(* Logix 5000 project; controller Amvex_Thorpe_Flowmeter vendor 1 type 14 code 106 rev 33.13; software revision 33.01; part 14 of 16 *)
(* tags used below, declared in another part *)
   Barcode_Result_DATA : SINT[128];
   HMI_Counter_ONS : BOOL;
   IV3_Prog_AOI : IvSwichPrgoram;
   Part_count : DINT;
   Prog_Switch_ons : BOOL;
   SR_Read_Request : BOOL;
   Test : Connect;
   Alicat_Status_ONS : BOOL[32];
   Barcode_timeout : TIMER;
   Cycle_Count_Ctr : COUNTER;
   Cycle_Count_ONS : BOOL;
   Cycle_Time_ONS : BOOL;
   FIRST_SCAN : BOOL;
   HMI : HMI_Temp;
   MCP : MCP;
   RCP1 : RCP1;
   RCP1_00 : UDT_ID0;
   Safety_OK : BOOL;
   Temp_Cycle_Time_Current : REAL;
   Temp_Cycle_Time_Last : REAL;
   Temp_Cycle_Timer : TIMER;
(* MCP_Main, continued *)

ROUTINE R09_IV3_VISION   (* ladder *)
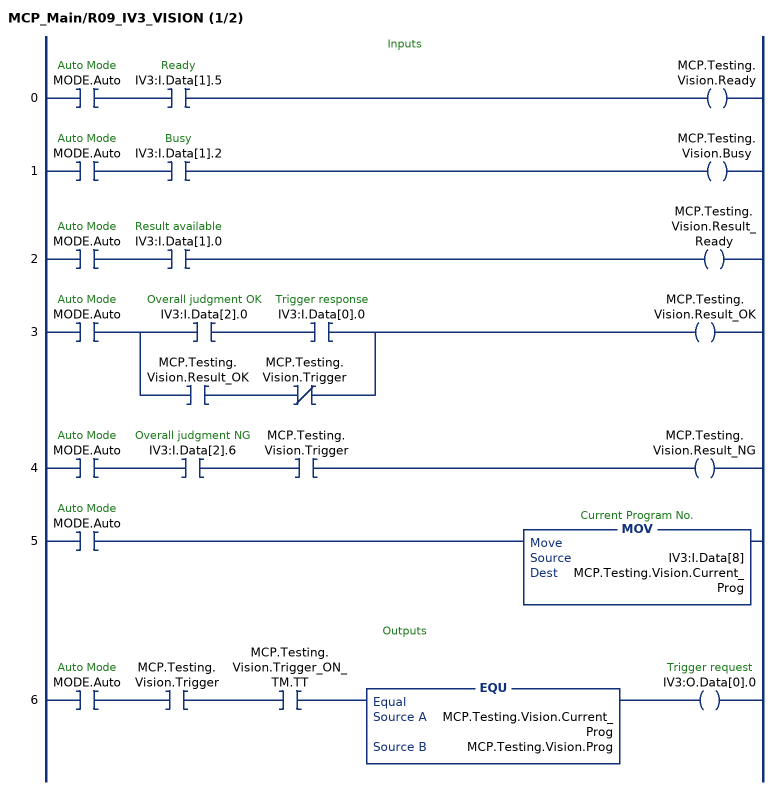
   // Inputs
   0: XIC(MODE.Auto)XIC(IV3:I.Data[1].5)OTE(MCP.Testing.Vision.Ready);
   1: XIC(MODE.Auto)XIC(IV3:I.Data[1].2)OTE(MCP.Testing.Vision.Busy);
   2: XIC(MODE.Auto)XIC(IV3:I.Data[1].0)OTE(MCP.Testing.Vision.Result_Ready);
   3: XIC(MODE.Auto)[XIC(IV3:I.Data[2].0) XIC(IV3:I.Data[0].0) ,XIC(MCP.Testing.Vision.Result_OK) XIO(MCP.Testing.Vision.Trigger) ]OTE(MCP.Testing.Vision.Result_OK);
   4: XIC(MODE.Auto)XIC(IV3:I.Data[2].6)XIC(MCP.Testing.Vision.Trigger)OTE(MCP.Testing.Vision.Result_NG);
   5: XIC(MODE.Auto)MOV(IV3:I.Data[8],MCP.Testing.Vision.Current_Prog);
   // Outputs
   6: XIC(MODE.Auto)XIC(MCP.Testing.Vision.Trigger)XIC(MCP.Testing.Vision.Trigger_ON_TM.TT)EQU(MCP.Testing.Vision.Current_Prog,MCP.Testing.Vision.Prog)OTE(IV3:O.Data[0].0);
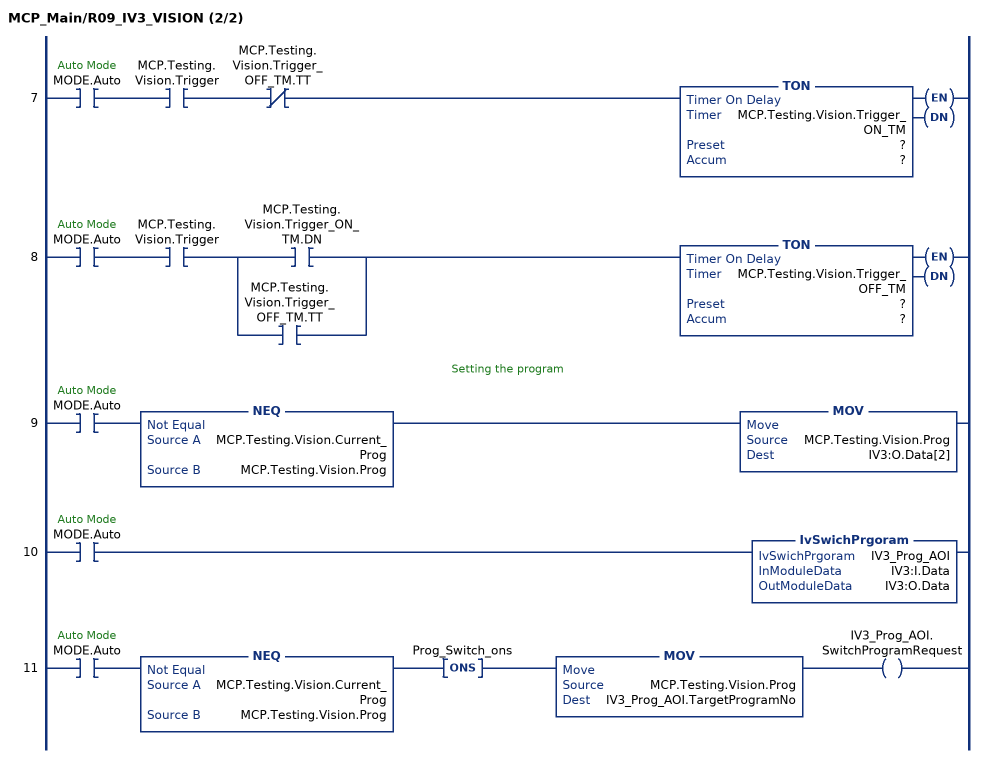
   7: XIC(MODE.Auto)XIC(MCP.Testing.Vision.Trigger)XIO(MCP.Testing.Vision.Trigger_OFF_TM.TT)TON(MCP.Testing.Vision.Trigger_ON_TM,?,?);
   8: XIC(MODE.Auto)XIC(MCP.Testing.Vision.Trigger)[XIC(MCP.Testing.Vision.Trigger_ON_TM.DN) ,XIC(MCP.Testing.Vision.Trigger_OFF_TM.TT) ]TON(MCP.Testing.Vision.Trigger_OFF_TM,?,?);
   // Setting the program
   9: XIC(MODE.Auto)NEQ(MCP.Testing.Vision.Current_Prog,MCP.Testing.Vision.Prog)MOV(MCP.Testing.Vision.Prog,IV3:O.Data[2]);
   10: XIC(MODE.Auto)IvSwichPrgoram(IV3_Prog_AOI,IV3:I.Data,IV3:O.Data);
   11: XIC(MODE.Auto)NEQ(MCP.Testing.Vision.Current_Prog,MCP.Testing.Vision.Prog)ONS(Prog_Switch_ons)MOV(MCP.Testing.Vision.Prog,IV3_Prog_AOI.TargetProgramNo)OTE(IV3_Prog_AOI.SwitchProgramRequest);
END_ROUTINE

ROUTINE R10_BARCODE   (* ladder *)
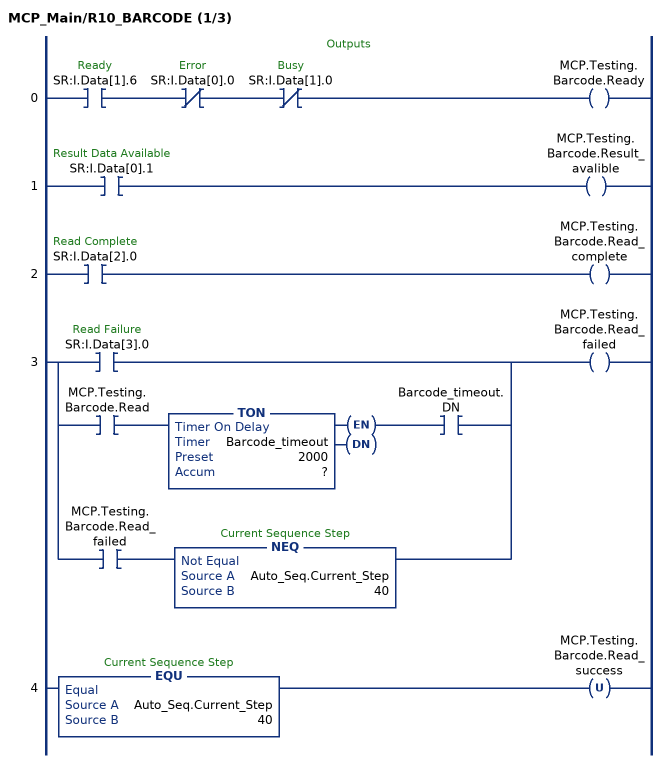
   // Outputs
   0: XIC(SR:I.Data[1].6)XIO(SR:I.Data[0].0)XIO(SR:I.Data[1].0)OTE(MCP.Testing.Barcode.Ready);
   1: XIC(SR:I.Data[0].1)OTE(MCP.Testing.Barcode.Result_avalible);
   2: XIC(SR:I.Data[2].0)OTE(MCP.Testing.Barcode.Read_complete);
   3: [XIC(SR:I.Data[3].0) ,XIC(MCP.Testing.Barcode.Read) TON(Barcode_timeout,?,?) XIC(Barcode_timeout.DN) ,XIC(MCP.Testing.Barcode.Read_failed) NEQ(Auto_Seq.Current_Step,40) ]OTE(MCP.Testing.Barcode.Read_failed);
   4: EQU(Auto_Seq.Current_Step,40)OTU(MCP.Testing.Barcode.Read_success);
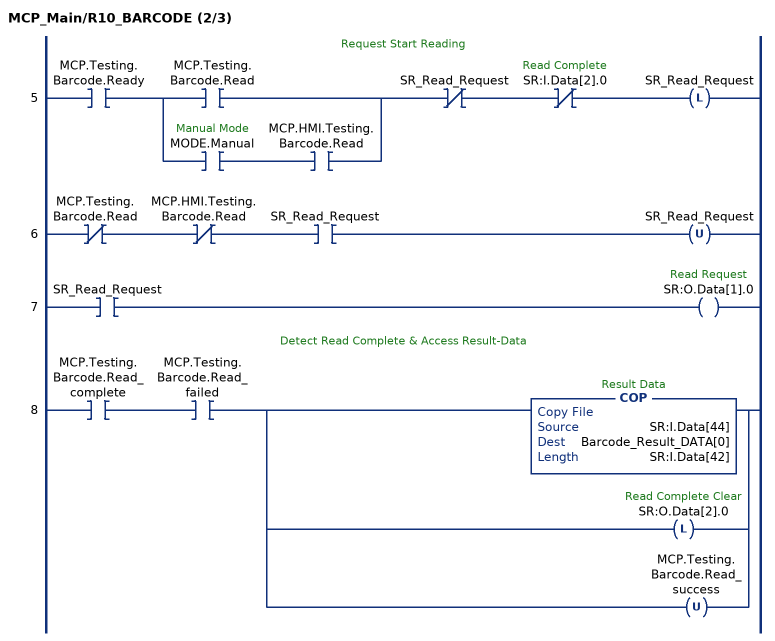
   // Request Start Reading
   5: XIC(MCP.Testing.Barcode.Ready)[XIC(MCP.Testing.Barcode.Read) ,XIC(MODE.Manual) XIC(MCP.HMI.Testing.Barcode.Read) ]XIO(SR_Read_Request)XIO(SR:I.Data[2].0)OTL(SR_Read_Request);
   6: XIO(MCP.Testing.Barcode.Read)XIO(MCP.HMI.Testing.Barcode.Read)XIC(SR_Read_Request)OTU(SR_Read_Request);
   7: XIC(SR_Read_Request)OTE(SR:O.Data[1].0);
   // Detect Read Complete & Access Result-Data
   8: XIC(MCP.Testing.Barcode.Read_complete)XIC(MCP.Testing.Barcode.Read_failed)[COP(SR:I.Data[44],Barcode_Result_DATA[0],SR:I.Data[42]) ,OTL(SR:O.Data[2].0) ,OTU(MCP.Testing.Barcode.Read_success) ];
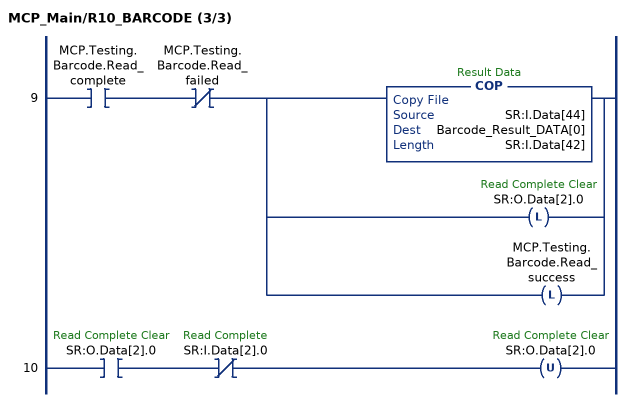
   9: XIC(MCP.Testing.Barcode.Read_complete)XIO(MCP.Testing.Barcode.Read_failed)[COP(SR:I.Data[44],Barcode_Result_DATA[0],SR:I.Data[42]) ,OTL(SR:O.Data[2].0) ,OTL(MCP.Testing.Barcode.Read_success) ];
   10: XIC(SR:O.Data[2].0)XIO(SR:I.Data[2].0)OTU(SR:O.Data[2].0);
END_ROUTINE

ROUTINE R11_VFD   (* ladder *)
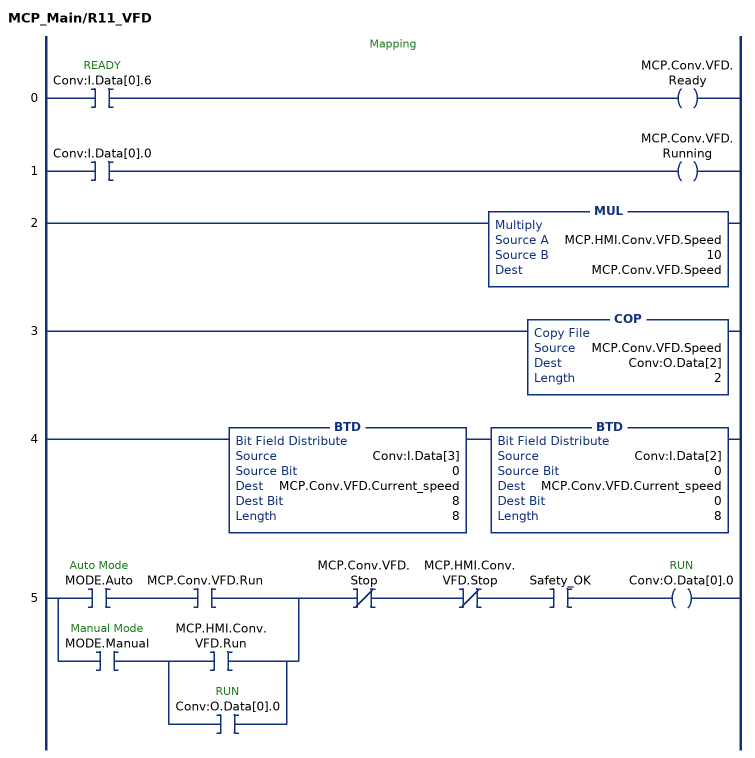
   // Mapping
   0: XIC(Conv:I.Data[0].6)OTE(MCP.Conv.VFD.Ready);
   1: XIC(Conv:I.Data[0].0)OTE(MCP.Conv.VFD.Running);
   2: MUL(MCP.HMI.Conv.VFD.Speed,10,MCP.Conv.VFD.Speed);
   3: COP(MCP.Conv.VFD.Speed,Conv:O.Data[2],2);
   4: BTD(Conv:I.Data[3],0,MCP.Conv.VFD.Current_speed,8,8)BTD(Conv:I.Data[2],0,MCP.Conv.VFD.Current_speed,0,8);
   5: [XIC(MODE.Auto) XIC(MCP.Conv.VFD.Run) ,XIC(MODE.Manual) [XIC(MCP.HMI.Conv.VFD.Run) ,XIC(Conv:O.Data[0].0) ] ]XIO(MCP.Conv.VFD.Stop)XIO(MCP.HMI.Conv.VFD.Stop)XIC(Safety_OK)OTE(Conv:O.Data[0].0);
END_ROUTINE

ROUTINE R12_HMI   (* ladder *)
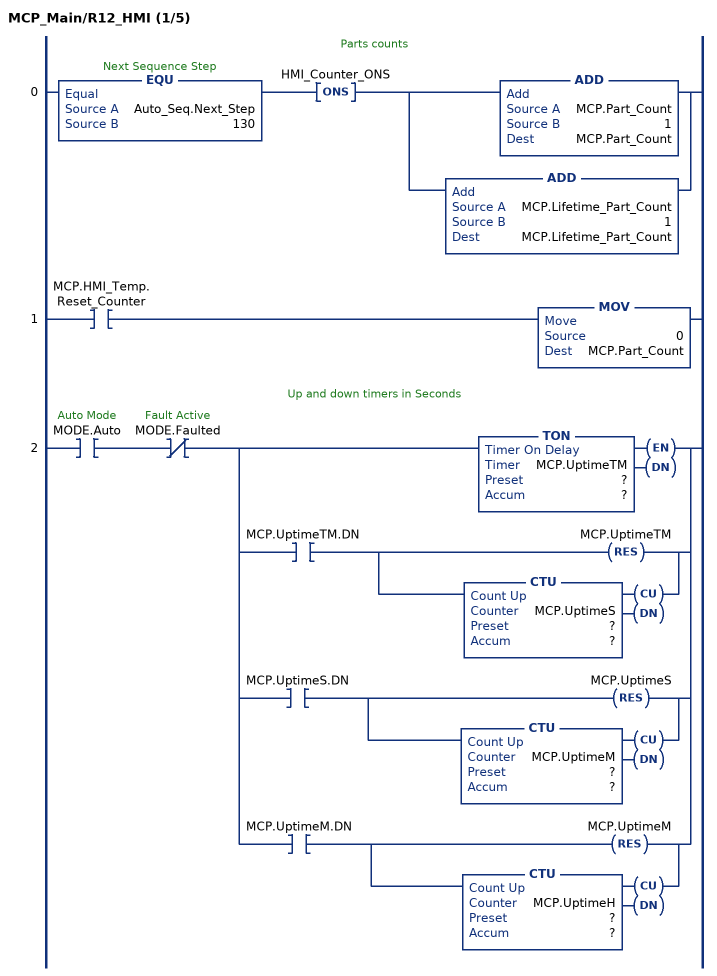
   // Parts counts
   0: EQU(Auto_Seq.Next_Step,130)ONS(HMI_Counter_ONS)[ADD(MCP.Part_Count,1,MCP.Part_Count) ,ADD(MCP.Lifetime_Part_Count,1,MCP.Lifetime_Part_Count) ];
   1: XIC(MCP.HMI_Temp.Reset_Counter)MOV(0,MCP.Part_Count);
   // Up and down timers in Seconds
   2: XIC(MODE.Auto)XIO(MODE.Faulted)[TON(MCP.UptimeTM,?,?) ,XIC(MCP.UptimeTM.DN) [RES(MCP.UptimeTM) ,CTU(MCP.UptimeS,?,?) ] ,XIC(MCP.UptimeS.DN) [RES(MCP.UptimeS) ,CTU(MCP.UptimeM,?,?) ] ,XIC(MCP.UptimeM.DN) [RES(MCP.UptimeM) ,CTU(MCP.UptimeH,?,?) ] ];
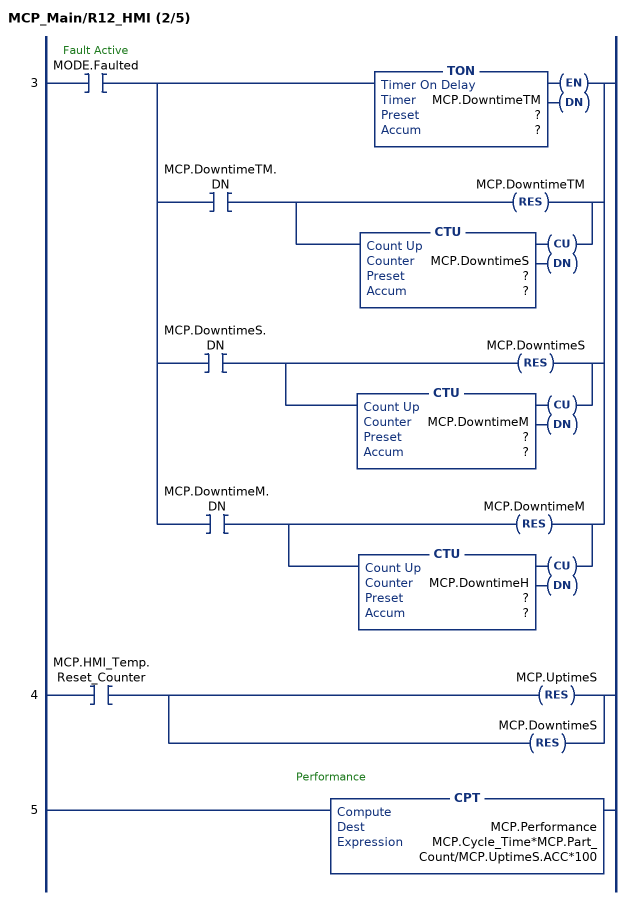
   3: XIC(MODE.Faulted)[TON(MCP.DowntimeTM,?,?) ,XIC(MCP.DowntimeTM.DN) [RES(MCP.DowntimeTM) ,CTU(MCP.DowntimeS,?,?) ] ,XIC(MCP.DowntimeS.DN) [RES(MCP.DowntimeS) ,CTU(MCP.DowntimeM,?,?) ] ,XIC(MCP.DowntimeM.DN) [RES(MCP.DowntimeM) ,CTU(MCP.DowntimeH,?,?) ] ];
   4: XIC(MCP.HMI_Temp.Reset_Counter)[RES(MCP.UptimeS) ,RES(MCP.DowntimeS) ];
   // Performance
   5: CPT(MCP.Performance,MCP.Cycle_Time*MCP.Part_Count/MCP.UptimeS.ACC*100);
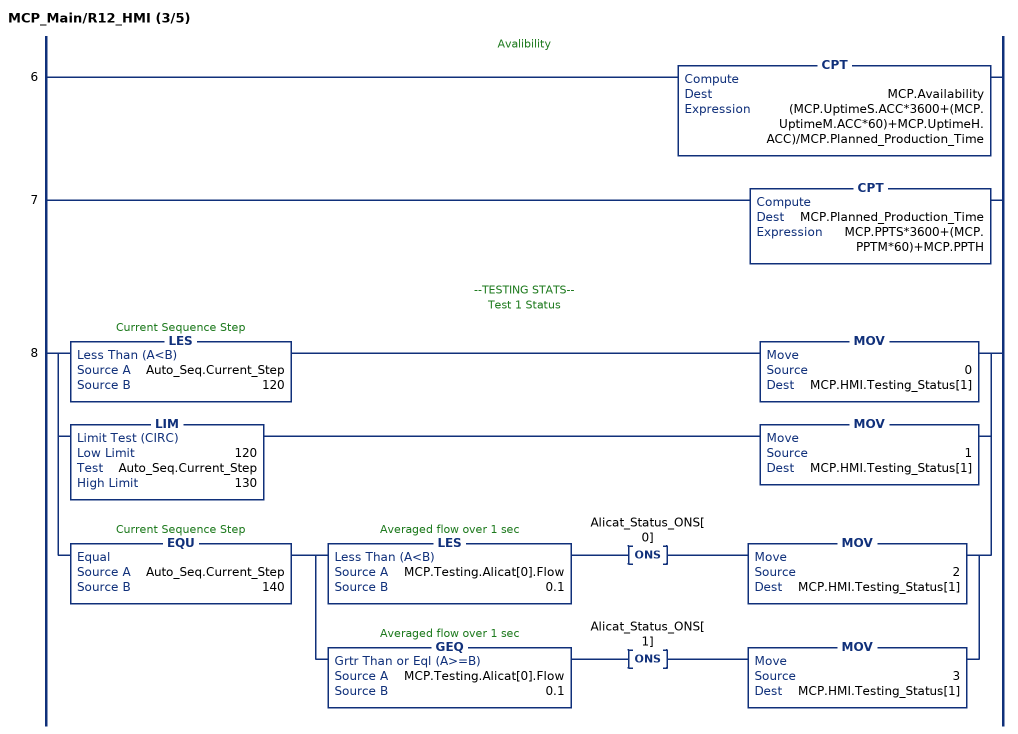
   // Avalibility
   6: CPT(MCP.Availability,(MCP.UptimeS.ACC*3600+(MCP.UptimeM.ACC*60)+MCP.UptimeH.ACC)/MCP.Planned_Production_Time);
   7: CPT(MCP.Planned_Production_Time,MCP.PPTS*3600+(MCP.PPTM*60)+MCP.PPTH);
   // --TESTING STATS--
   // Test 1 Status
   8: [LES(Auto_Seq.Current_Step,120) MOV(0,MCP.HMI.Testing_Status[1]) ,LIM(120,Auto_Seq.Current_Step,130) MOV(1,MCP.HMI.Testing_Status[1]) ,EQU(Auto_Seq.Current_Step,140) [LES(MCP.Testing.Alicat[0].Flow,0.1) ONS(Alicat_Status_ONS[0]) MOV(2,MCP.HMI.Testing_Status[1]) ,GEQ(MCP.Testing.Alicat[0].Flow,0.1) ONS(Alicat_Status_ONS[1]) MOV(3,MCP.HMI.Testing_Status[1]) ] ];
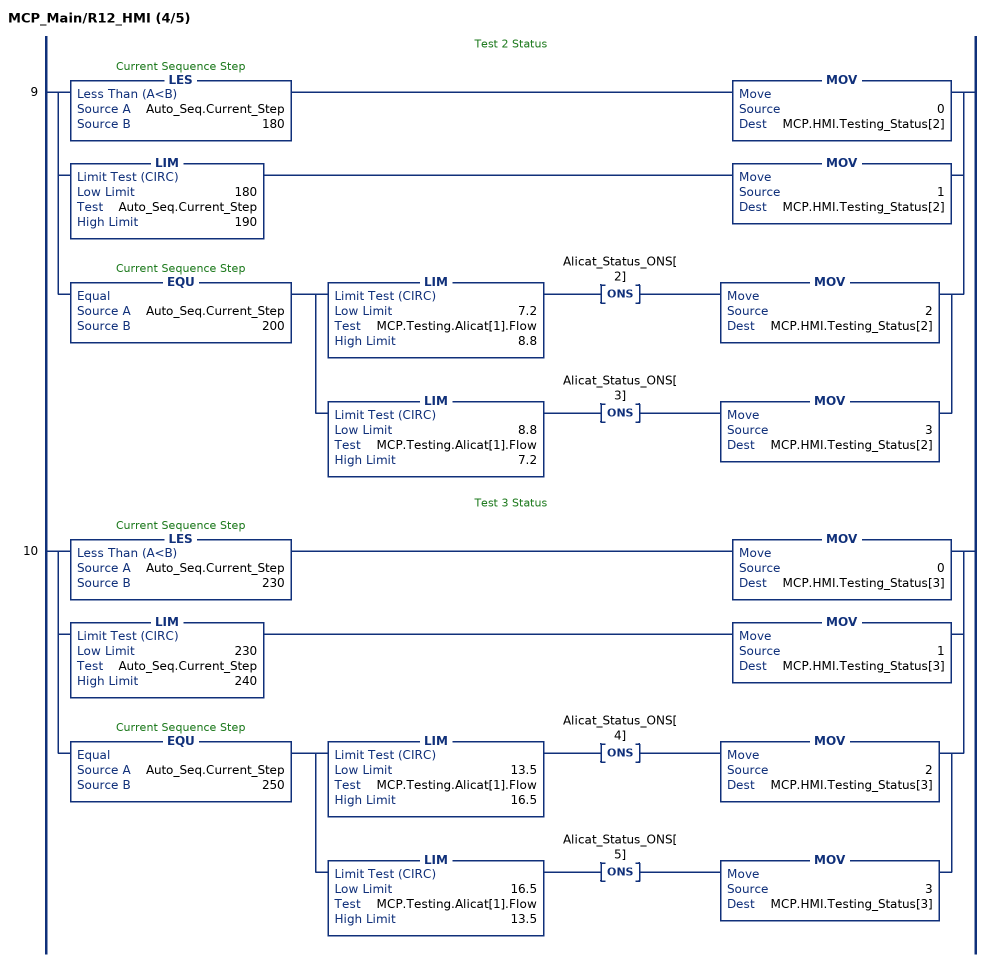
   // Test 2 Status
   9: [LES(Auto_Seq.Current_Step,180) MOV(0,MCP.HMI.Testing_Status[2]) ,LIM(180,Auto_Seq.Current_Step,190) MOV(1,MCP.HMI.Testing_Status[2]) ,EQU(Auto_Seq.Current_Step,200) [LIM(7.2,MCP.Testing.Alicat[1].Flow,8.8) ONS(Alicat_Status_ONS[2]) MOV(2,MCP.HMI.Testing_Status[2]) ,LIM(8.8,MCP.Testing.Alicat[1].Flow,7.2) ONS(Alicat_Status_ONS[3]) MOV(3,MCP.HMI.Testing_Status[2]) ] ];
   // Test 3 Status
   10: [LES(Auto_Seq.Current_Step,230) MOV(0,MCP.HMI.Testing_Status[3]) ,LIM(230,Auto_Seq.Current_Step,240) MOV(1,MCP.HMI.Testing_Status[3]) ,EQU(Auto_Seq.Current_Step,250) [LIM(13.5,MCP.Testing.Alicat[1].Flow,16.5) ONS(Alicat_Status_ONS[4]) MOV(2,MCP.HMI.Testing_Status[3]) ,LIM(16.5,MCP.Testing.Alicat[1].Flow,13.5) ONS(Alicat_Status_ONS[5]) MOV(3,MCP.HMI.Testing_Status[3]) ] ];
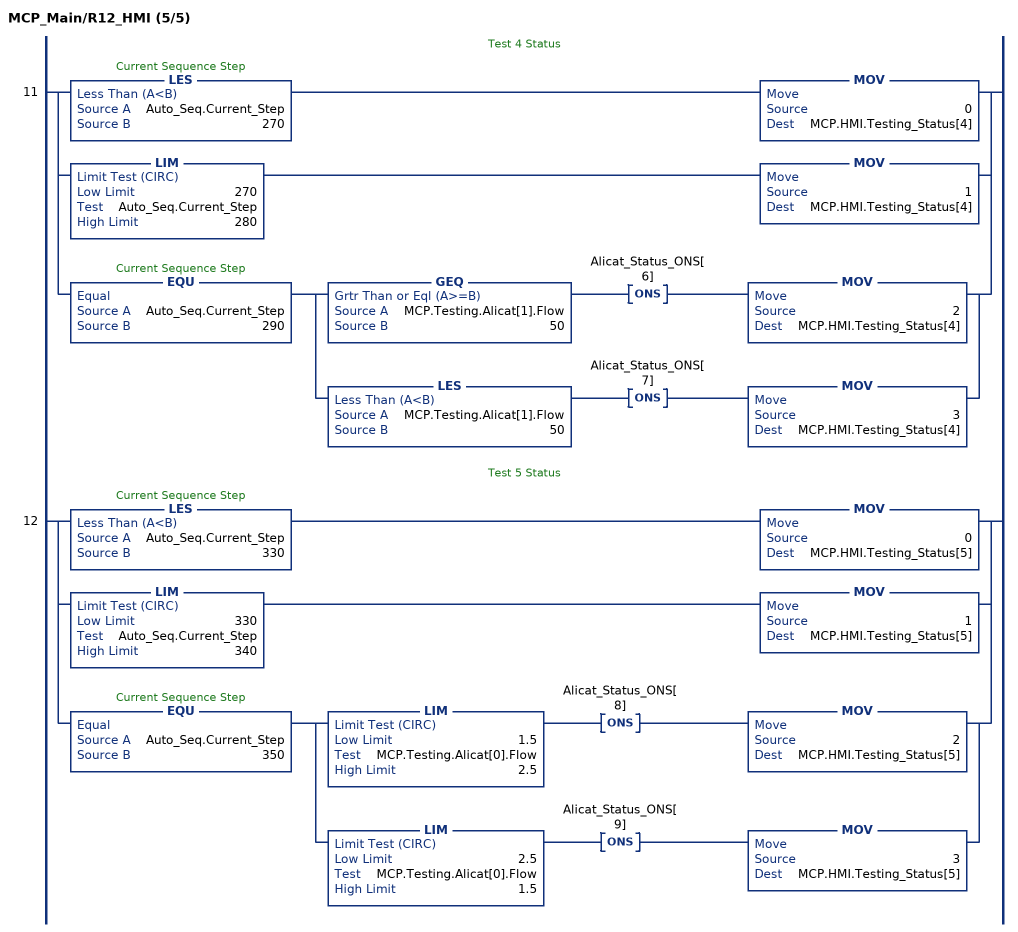
   // Test 4 Status
   11: [LES(Auto_Seq.Current_Step,270) MOV(0,MCP.HMI.Testing_Status[4]) ,LIM(270,Auto_Seq.Current_Step,280) MOV(1,MCP.HMI.Testing_Status[4]) ,EQU(Auto_Seq.Current_Step,290) [GEQ(MCP.Testing.Alicat[1].Flow,50) ONS(Alicat_Status_ONS[6]) MOV(2,MCP.HMI.Testing_Status[4]) ,LES(MCP.Testing.Alicat[1].Flow,50) ONS(Alicat_Status_ONS[7]) MOV(3,MCP.HMI.Testing_Status[4]) ] ];
   // Test 5 Status
   12: [LES(Auto_Seq.Current_Step,330) MOV(0,MCP.HMI.Testing_Status[5]) ,LIM(330,Auto_Seq.Current_Step,340) MOV(1,MCP.HMI.Testing_Status[5]) ,EQU(Auto_Seq.Current_Step,350) [LIM(1.5,MCP.Testing.Alicat[0].Flow,2.5) ONS(Alicat_Status_ONS[8]) MOV(2,MCP.HMI.Testing_Status[5]) ,LIM(2.5,MCP.Testing.Alicat[0].Flow,1.5) ONS(Alicat_Status_ONS[9]) MOV(3,MCP.HMI.Testing_Status[5]) ] ];
END_ROUTINE

ROUTINE R13_DATABASE   (* ladder *)
END_ROUTINE

ROUTINE R14_MODE   (* ladder *)
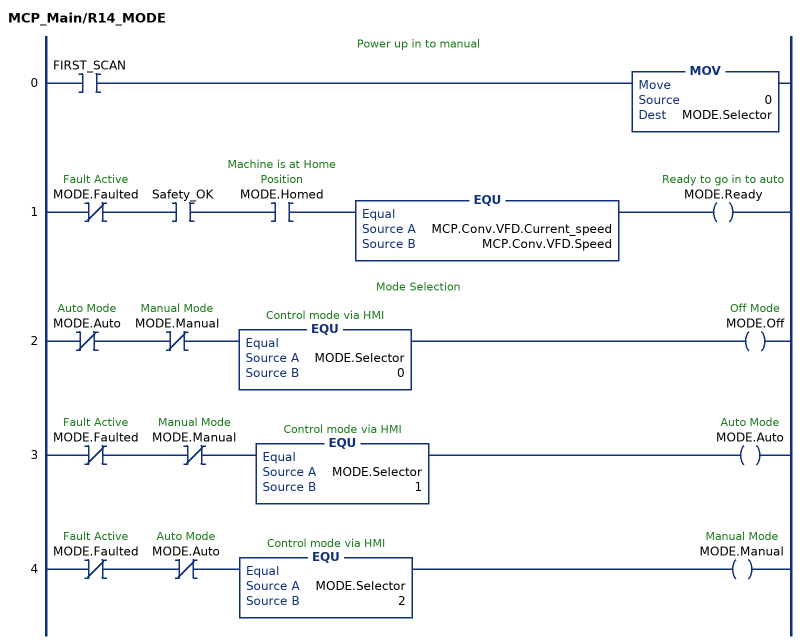
   // Power up in to manual
   0: XIC(FIRST_SCAN)MOV(0,MODE.Selector);
   1: XIO(MODE.Faulted)XIC(Safety_OK)XIC(MODE.Homed)EQU(MCP.Conv.VFD.Current_speed,MCP.Conv.VFD.Speed)OTE(MODE.Ready);
   // Mode Selection
   2: XIO(MODE.Auto)XIO(MODE.Manual)EQU(MODE.Selector,0)OTE(MODE.Off);
   3: XIO(MODE.Faulted)XIO(MODE.Manual)EQU(MODE.Selector,1)OTE(MODE.Auto);
   4: XIO(MODE.Faulted)XIO(MODE.Auto)EQU(MODE.Selector,2)OTE(MODE.Manual);
END_ROUTINE

ROUTINE R16_PROD_CNTR   (* ladder *)
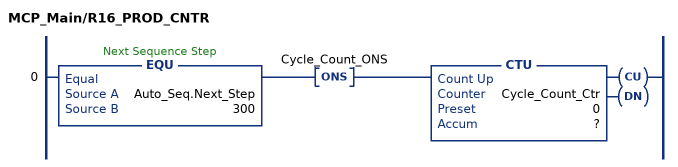
   0: EQU(Auto_Seq.Next_Step,300)ONS(Cycle_Count_ONS)CTU(Cycle_Count_Ctr,?,?);
END_ROUTINE

ROUTINE R17_CYCLE_TIME   (* ladder *)
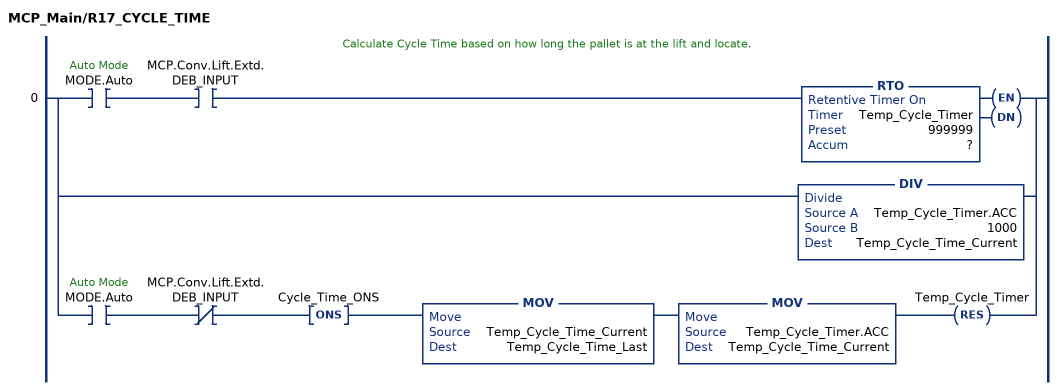
   // Calculate Cycle Time based on how long the pallet is at the lift and locate.
   0: [XIC(MODE.Auto) XIC(MCP.Conv.Lift.Extd.DEB_INPUT) RTO(Temp_Cycle_Timer,?,?) ,DIV(Temp_Cycle_Timer.ACC,1000,Temp_Cycle_Time_Current) ,XIC(MODE.Auto) XIO(MCP.Conv.Lift.Extd.DEB_INPUT) ONS(Cycle_Time_ONS) MOV(Temp_Cycle_Time_Current,Temp_Cycle_Time_Last) MOV(Temp_Cycle_Timer.ACC,Temp_Cycle_Time_Current) RES(Temp_Cycle_Timer) ];
END_ROUTINE

ROUTINE R18_HOME   (* ladder *)
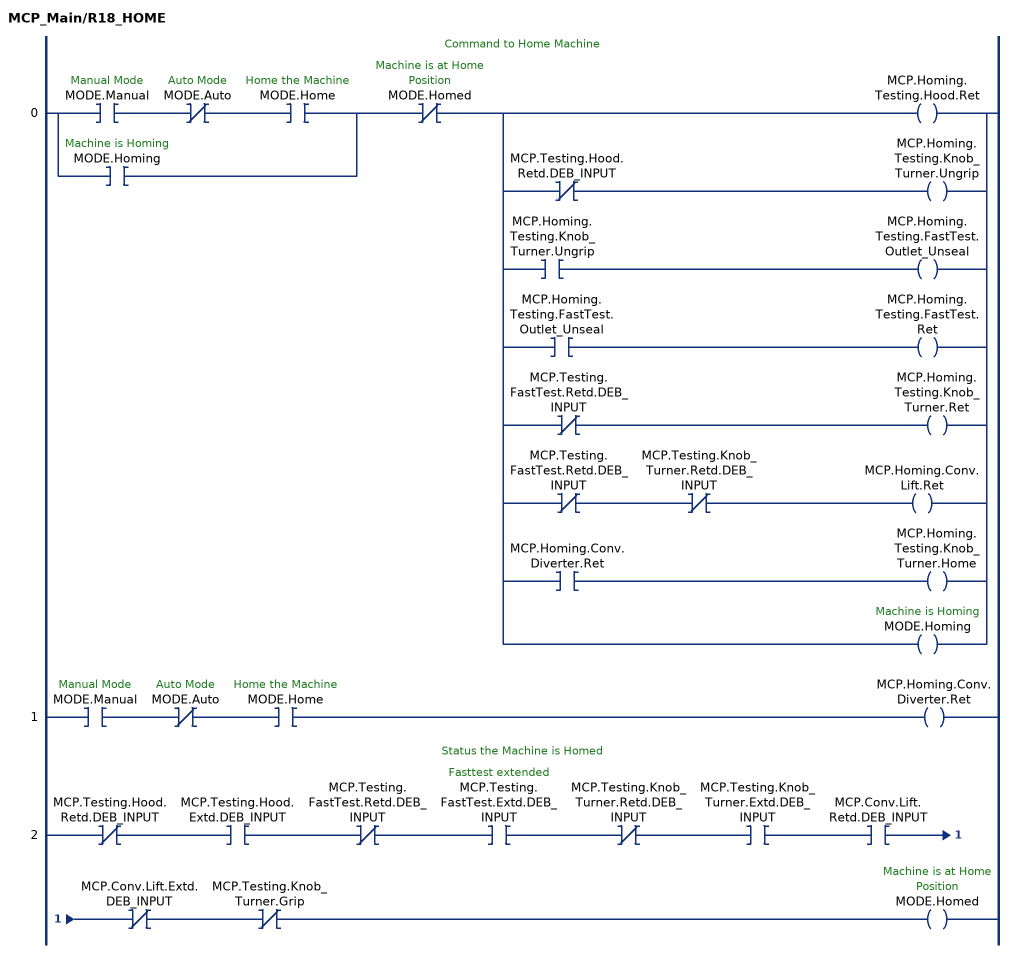
   // Command to Home Machine
   0: [XIC(MODE.Manual) XIO(MODE.Auto) XIC(MODE.Home) ,XIC(MODE.Homing) ]XIO(MODE.Homed)[OTE(MCP.Homing.Testing.Hood.Ret) ,XIO(MCP.Testing.Hood.Retd.DEB_INPUT) OTE(MCP.Homing.Testing.Knob_Turner.Ungrip) ,XIC(MCP.Homing.Testing.Knob_Turner.Ungrip) OTE(MCP.Homing.Testing.FastTest.Outlet_Unseal) ,XIC(MCP.Homing.Testing.FastTest.Outlet_Unseal) OTE(MCP.Homing.Testing.FastTest.Ret) ,XIO(MCP.Testing.FastTest.Retd.DEB_INPUT) OTE(MCP.Homing.Testing.Knob_Turner.Ret) ,XIO(MCP.Testing.FastTest.Retd.DEB_INPUT) XIO(MCP.Testing.Knob_Turner.Retd.DEB_INPUT) OTE(MCP.Homing.Conv.Lift.Ret) ,XIC(MCP.Homing.Conv.Diverter.Ret) OTE(MCP.Homing.Testing.Knob_Turner.Home) ,OTE(MODE.Homing) ];
   1: XIC(MODE.Manual)XIO(MODE.Auto)XIC(MODE.Home)OTE(MCP.Homing.Conv.Diverter.Ret);
   // Status the Machine is Homed
   2: XIO(MCP.Testing.Hood.Retd.DEB_INPUT)XIC(MCP.Testing.Hood.Extd.DEB_INPUT)XIO(MCP.Testing.FastTest.Retd.DEB_INPUT)XIC(MCP.Testing.FastTest.Extd.DEB_INPUT)XIO(MCP.Testing.Knob_Turner.Retd.DEB_INPUT)XIC(MCP.Testing.Knob_Turner.Extd.DEB_INPUT)XIC(MCP.Conv.Lift.Retd.DEB_INPUT)XIO(MCP.Conv.Lift.Extd.DEB_INPUT)XIO(MCP.Testing.Knob_Turner.Grip)OTE(MODE.Homed);
END_ROUTINE
END_PROGRAM

PROGRAM RPC1_Main   (* main routine MAIN *)
VAR
   Auto_Seq : SEQ := (Time_Out.PRE := 180000, Time_Out.ACC := 114179, Time_Out.EN := 1, Time_Out.TT := 1, Time_Out_Sec := 180);
   Clear_TM : TIMER := (PRE := 500);
   Counter_ONS : BOOL;
   DriveTime_TM : TIMER := (PRE := 7000);
   FAULT : DINT;
   FAULTED : DINT;
   Flash_Timer_Off : TIMER := (PRE := 500, ACC := 250, EN := 1, TT := 1);
   Flash_Timer_On : TIMER := (PRE := 500);
   MODE : MODE := (Off := 1, Faulted := 1);
   nullString : STRING;
   RCD_ONS : BOOL;
   RESET : BOOL;
   RESET_ONS : BOOL;
   StringFix : CONTROL := (LEN := 20);
   StringFix_ONS : BOOL;
END_VAR

ROUTINE MAIN   (* ladder *)
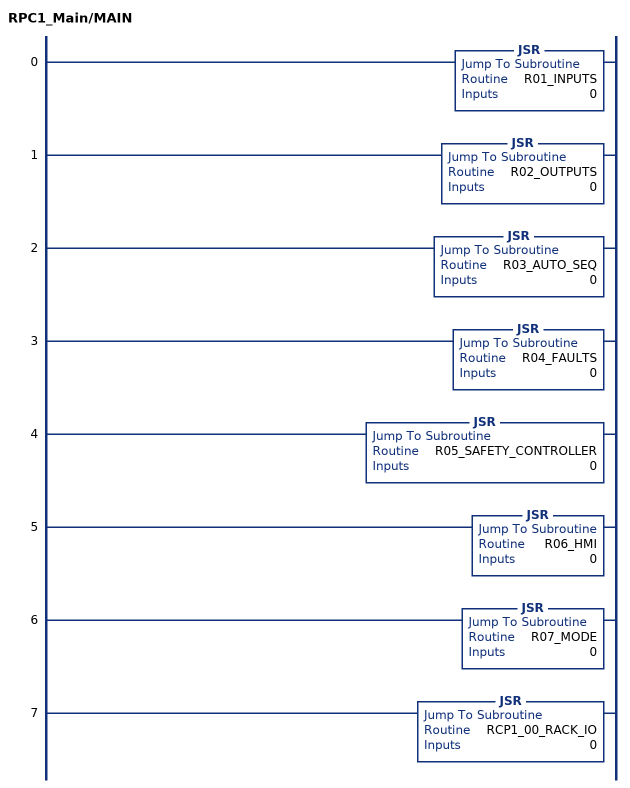
   0: JSR(R01_INPUTS,0);
   1: JSR(R02_OUTPUTS,0);
   2: JSR(R03_AUTO_SEQ,0);
   3: JSR(R04_FAULTS,0);
   4: JSR(R05_SAFETY_CONTROLLER,0);
   5: JSR(R06_HMI,0);
   6: JSR(R07_MODE,0);
   7: JSR(RCP1_00_RACK_IO,0);
END_ROUTINE

ROUTINE R01_INPUTS   (* ladder *)
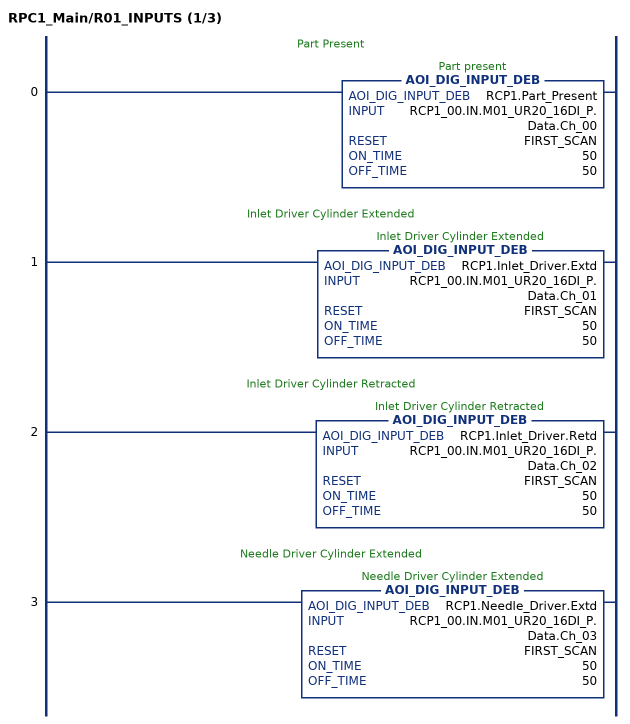
   // Part Present
   0: AOI_DIG_INPUT_DEB(RCP1.Part_Present,RCP1_00.IN.M01_UR20_16DI_P.Data.Ch_00,FIRST_SCAN,50,50);
   // Inlet Driver Cylinder Extended
   1: AOI_DIG_INPUT_DEB(RCP1.Inlet_Driver.Extd,RCP1_00.IN.M01_UR20_16DI_P.Data.Ch_01,FIRST_SCAN,50,50);
   // Inlet Driver Cylinder Retracted
   2: AOI_DIG_INPUT_DEB(RCP1.Inlet_Driver.Retd,RCP1_00.IN.M01_UR20_16DI_P.Data.Ch_02,FIRST_SCAN,50,50);
   // Needle Driver Cylinder Extended
   3: AOI_DIG_INPUT_DEB(RCP1.Needle_Driver.Extd,RCP1_00.IN.M01_UR20_16DI_P.Data.Ch_03,FIRST_SCAN,50,50);
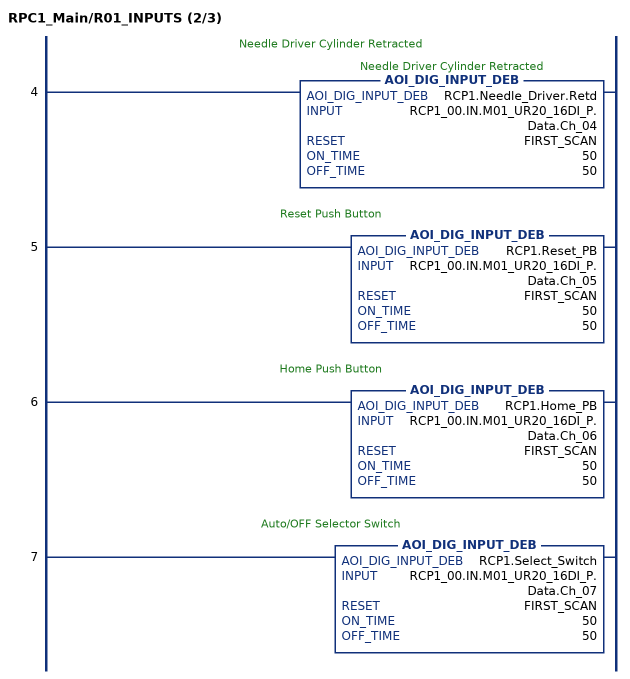
   // Needle Driver Cylinder Retracted
   4: AOI_DIG_INPUT_DEB(RCP1.Needle_Driver.Retd,RCP1_00.IN.M01_UR20_16DI_P.Data.Ch_04,FIRST_SCAN,50,50);
   // Reset Push Button
   5: AOI_DIG_INPUT_DEB(RCP1.Reset_PB,RCP1_00.IN.M01_UR20_16DI_P.Data.Ch_05,FIRST_SCAN,50,50);
   // Home Push Button
   6: AOI_DIG_INPUT_DEB(RCP1.Home_PB,RCP1_00.IN.M01_UR20_16DI_P.Data.Ch_06,FIRST_SCAN,50,50);
   // Auto/OFF Selector Switch
   7: AOI_DIG_INPUT_DEB(RCP1.Select_Switch,RCP1_00.IN.M01_UR20_16DI_P.Data.Ch_07,FIRST_SCAN,50,50);
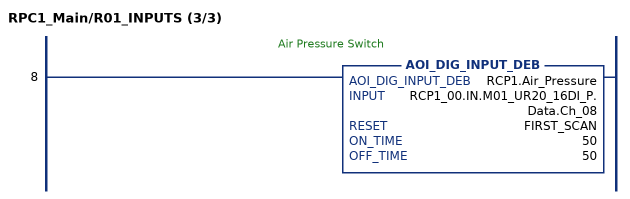
   // Air Pressure Switch
   8: AOI_DIG_INPUT_DEB(RCP1.Air_Pressure,RCP1_00.IN.M01_UR20_16DI_P.Data.Ch_08,FIRST_SCAN,50,50);
END_ROUTINE
